% RSLogix 500 project P1_PSI-Level.RSS, saved by version 8.30.00.16 %
PROJECT "UNTITLED"    % processor: Bul.1763 MicroLogix 1100 Series B %

PROGRAM FILES
  LAD 2 "MAIN"  3 rungs
  LAD 3 "IO"  5 rungs
  LAD 4 "CTRL LOGIC"  11 rungs

DATA FILES
  O0 OUTPUT  5 elements
  I1 INPUT  7 elements
  S2 STATUS  66 elements
  B3 BINARY  1 elements
  T4 TIMER  4 elements
  C5 COUNTER  1 elements
  R6 CONTROL  1 elements
  N7 INTEGER  1 elements
  F8 FLOAT  1 elements

LADDER 2 "MAIN"
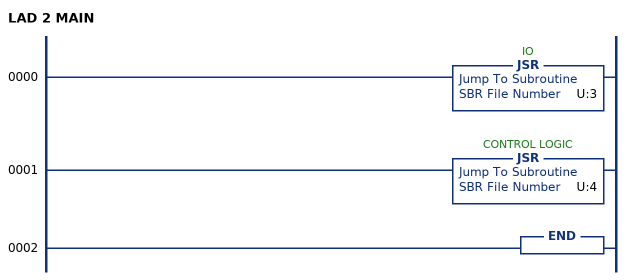
% Rung: 0 %
SOR JSR U:3 EOR
%   U:3  "IO" %
% Rung: 1 %
SOR JSR U:4 EOR
%   U:4  "CONTROL LOGIC" %
% Rung: 2 %
SOR END EOR

LADDER 3 "IO"
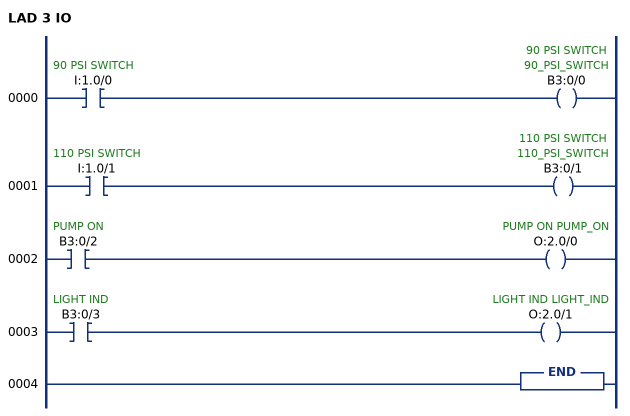
% Rung: 0 %
SOR XIC I:1.0/0 OTE B3:0/0 EOR
%   I:1.0/0  "90 PSI SWITCH" %
%   B3:0/0  90_PSI_SWITCH  "90 PSI SWITCH" %
% Rung: 1 %
SOR XIC I:1.0/1 OTE B3:0/1 EOR
%   I:1.0/1  "110 PSI SWITCH" %
%   B3:0/1  110_PSI_SWITCH  "110 PSI SWITCH" %
% Rung: 2 %
SOR XIC B3:0/2 OTE O:2.0/0 EOR
%   B3:0/2  "PUMP ON" %
%   O:2.0/0  PUMP_ON  "PUMP ON" %
% Rung: 3 %
SOR XIC B3:0/3 OTE O:2.0/1 EOR
%   B3:0/3  "LIGHT IND" %
%   O:2.0/1  LIGHT_IND  "LIGHT IND" %
% Rung: 4 %
SOR END EOR

LADDER 4 "CTRL LOGIC"
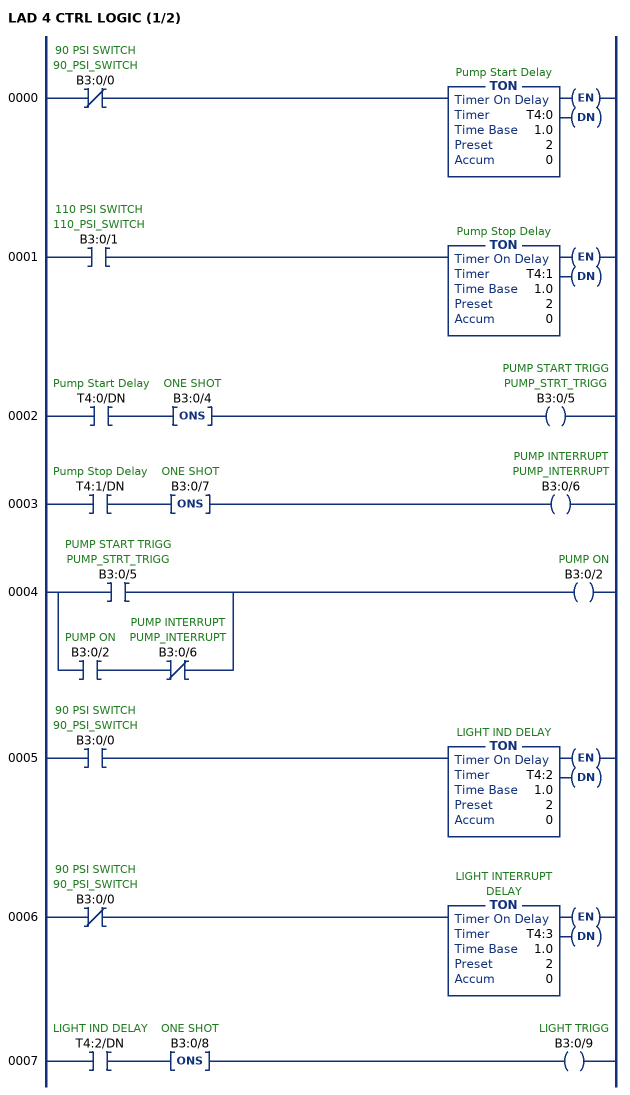
% Rung: 0 %
SOR XIO B3:0/0 TON T4:0 1.0 2 0 EOR
%   B3:0/0  90_PSI_SWITCH  "90 PSI SWITCH" %
%   T4:0  "Pump Start Delay" %
% Rung: 1 %
SOR XIC B3:0/1 TON T4:1 1.0 2 0 EOR
%   B3:0/1  110_PSI_SWITCH  "110 PSI SWITCH" %
%   T4:1  "Pump Stop Delay" %
% Rung: 2 %
SOR XIC T4:0/DN ONS B3:0/4 OTE B3:0/5 EOR
%   T4:0  "Pump Start Delay" %
%   B3:0/4  "ONE SHOT" %
%   B3:0/5  PUMP_STRT_TRIGG  "PUMP START TRIGG" %
% Rung: 3 %
SOR XIC T4:1/DN ONS B3:0/7 OTE B3:0/6 EOR
%   T4:1  "Pump Stop Delay" %
%   B3:0/7  "ONE SHOT" %
%   B3:0/6  PUMP_INTERRUPT  "PUMP INTERRUPT" %
% Rung: 4 %
SOR BST XIC B3:0/5 NXB XIC B3:0/2 XIO B3:0/6 BND OTE B3:0/2 EOR
%   B3:0/5  PUMP_STRT_TRIGG  "PUMP START TRIGG" %
%   B3:0/2  "PUMP ON" %
%   B3:0/6  PUMP_INTERRUPT  "PUMP INTERRUPT" %
% Rung: 5 %
SOR XIC B3:0/0 TON T4:2 1.0 2 0 EOR
%   B3:0/0  90_PSI_SWITCH  "90 PSI SWITCH" %
%   T4:2  "LIGHT IND DELAY" %
% Rung: 6 %
SOR XIO B3:0/0 TON T4:3 1.0 2 0 EOR
%   B3:0/0  90_PSI_SWITCH  "90 PSI SWITCH" %
%   T4:3  "LIGHT INTERRUPT DELAY" %
% Rung: 7 %
SOR XIC T4:2/DN ONS B3:0/8 OTE B3:0/9 EOR
%   T4:2  "LIGHT IND DELAY" %
%   B3:0/8  "ONE SHOT" %
%   B3:0/9  "LIGHT TRIGG" %

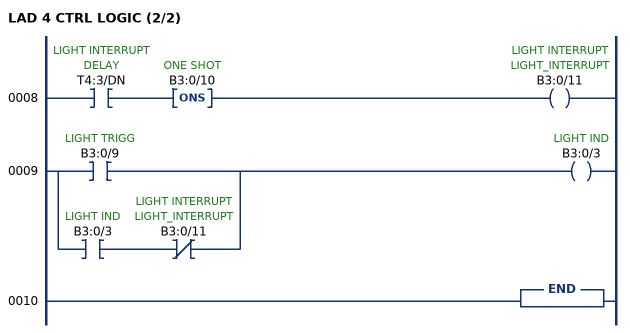
% Rung: 8 %
SOR XIC T4:3/DN ONS B3:0/10 OTE B3:0/11 EOR
%   T4:3  "LIGHT INTERRUPT DELAY" %
%   B3:0/10  "ONE SHOT" %
%   B3:0/11  LIGHT_INTERRUPT  "LIGHT INTERRUPT" %
% Rung: 9 %
SOR BST XIC B3:0/9 NXB XIC B3:0/3 XIO B3:0/11 BND OTE B3:0/3 EOR
%   B3:0/9  "LIGHT TRIGG" %
%   B3:0/3  "LIGHT IND" %
%   B3:0/11  LIGHT_INTERRUPT  "LIGHT INTERRUPT" %
% Rung: 10 %
SOR END EOR

OTHER DOCUMENTED ADDRESSES
  T4:0/0  "Pump Start Delay"
  T4:0/1  "Pump Stop Delay"

DATA TABLE (non-zero values as saved)
DATA T4
% .PRE .ACC %
% T4:0 % 2 0
% T4:1 % 2 0
% T4:2 % 2 0
% T4:3 % 2 0
